{attribute 'GeneratedUsingTerminal: EL9550-0010-0016'}
{attribute addProperty BoxType "EL9550-0010-0016"}
{attribute addProperty Id "UndervoltageAT %I*BOOL1OvervoltageAT %I*BOOL1"}
{attribute addProperty CRC "3677696296"}
{attribute addProperty Size "2"}
TYPE Status_Us_DB353128 :
STRUCT
	{attribute addProperty Name "Undervoltage"}
	Undervoltage AT %I* : BOOL;
	{attribute addProperty Name "Overvoltage"}
	Overvoltage AT %I* : BOOL;
END_STRUCT
END_TYPE

(* stored: Version 1.2.0.0, ProductVersion 3.1.4024.9
   DUT Status_Us_DB353128: Id {4ae783fd-d03b-43bd-bb40-a8ec6751f2c2} *)
